(* CODESYS project e!C_Integration_Test_2.ECP

Project tree, tasks and I/O mapping:
  PFC_8206_PRO : 750-8206 PFC200 2ETH RS CAN DPS, WAGO, order no. 0750-8206, version 5.11.1.16
    application Application
      libraries: Util, * (System)
      task PLC_Task (cyclic, interval t#10ms, priority 14) calls PLC_PRG
      task VISU_TASK (cyclic, interval 100 ms, priority 15) calls VisuElems.Visu_Prg
      program PLC_PRG [ST]: Test2
      global variables NVL1_From8206
      declarations NVL1_From8203
      MODBUS/
        data type typFC_352_tcp
      global variables MODBUS
      visualisation Visu1
      image pool ImagePool8206
      global variables GNVL_RW_1
    DeviceAdapter
    Kbus : Kbus, WAGO, version 1.4.0.2
        unmapped channels: K-BUS diagnostics
      _8DI_8DO_24V_DC_0_5A : 0750-1506, WAGO, order no. 0750-1506, version 0.0.0.11
          settings: K-BUS Module slot index = 1
          input  LocalIn_Byte_1 AT %IB0 : BYTE  // _IN
          output LocalOut_Byte_1 AT %QB0 : BYTE  // _OUT
        DeviceAdapter
    MODBUS
      MODBUS : MODBUS, WAGO, order no. n/a, version 1.1.1.15
        _internal_1006_0001_Master : MODBUS Master, WAGO, order no. n/a, version 1.1.1.15
          _internal_1006_0001_IP : MODBUS IP Interface, WAGO, order no. n/a, version 1.1.1.15
              settings: IP settings.Address = '192.168.1.8'; Minimum Request Interval = 0 ms
            _internal_1006_0001_Remote_Slave : MODBUS Remote Slave, WAGO, order no. n/a, version 1.1.1.15
                settings: GeneratedChannel 100005.Cycle Time = 200 ms; GeneratedChannel 100005.Write Address = 512 Registers or Coils; GeneratedChannel 100005.Write Length = 1 Registers or Coils; Offset 100010 = 0; Slave address / Unit identifier = 1
                output Application.MODBUS.FC_352_tcp.dOut_1 : BOOL  // Mapping100020
    PROFIBUS
      PROFIBUS : PROFIBUS, WAGO, version 1.0.0.0
          settings: DT_Slot1_std:ARRAY[0..9] OF BYTE = 40; CT_Slot1_std:ARRAY[0..9] OF BYTE = 2; DT_Slot2_std:ARRAY[0..9] OF BYTE = 40; CT_Slot2_std:ARRAY[0..9] OF BYTE = 1
          input  To8206_ByteArray_1 : ARRAY[0..9] OF BYTE  // Slot1
          output From8206_ByteArray_1 : ARRAY[0..9] OF BYTE  // Slot2
    CANbus
      WAGO_CANopen_Manager : WAGO CANopen Manager, WAGO, version 3.5.4.10
          settings: ConfigVersion = 50659584
        _750_347m_V14 : 750-347m_V14, WAGO, order no. 750-347, version Revision=16#00000001, FileVersion=1.14
            settings: General Options.Reset Node = false; NODEIDSAVED = 4; SDO Timeout = 1000000; SubIndex for reset node = 0; Emergency-General Parameters.Emergency COBID = 16#00000084; Settings.COBID = 16#00000204; Settings.Transmission Type = 16#FF; Settings.available PDO-Parameter.Inhibit Time available = FALSE; Settings.available PDO-Parameter.Event Timer available = FALSE; Settings.Inhibit Time = 0; Settings.Event Timer = 0; Generic COBID = '$NODEID+16#0200'; Process by CANopenManager = TRUE; Settings.COBID = 16#00000184; Settings.Transmission Type = 16#FF; Settings.available PDO-Parameter.Inhibit Time available = TRUE; Settings.available PDO-Parameter.Event Timer available = TRUE; Settings.Inhibit Time = 0; Settings.Event Timer = 0; Generic COBID = '$NODEID+16#0180'; Process by CANopenManager = TRUE; WriteOutput8Bit : _75x_504_1.Index = 16#6200; WriteOutput8Bit : _75x_504_1.Subindex = 16#01; WriteOutput8Bit : _75x_504_1.ObjectLength = 8; ReadAnalogueInput16Bit : _75x_455_1.Index = 16#6401; ReadAnalogueInput16Bit : _75x_455_1.Subindex = 16#01; ReadAnalogueInput16Bit : _75x_455_1.ObjectLength = 16; ReadAnalogueInput16Bit : _75x_455_1.Index = 16#6401; ReadAnalogueInput16Bit : _75x_455_1.Subindex = 16#02; ReadAnalogueInput16Bit : _75x_455_1.ObjectLength = 16; ReadAnalogueInput16Bit : _75x_455_1.Index = 16#6401; ReadAnalogueInput16Bit : _75x_455_1.Subindex = 16#03; ReadAnalogueInput16Bit : _75x_455_1.ObjectLength = 16; ReadAnalogueInput16Bit : _75x_455_1.Index = 16#6401; ReadAnalogueInput16Bit : _75x_455_1.Subindex = 16#04; ReadAnalogueInput16Bit : _75x_455_1.ObjectLength = 16; SDO List.Set Guardtime.Index = 16#100C; SDO List.Set Guardtime.Subindex = 16#00; SDO List.Set Guardtime.Value = 16#00000000; SDO List.Set Guardtime.Size = 16;
              SDO List.Set Guardtime.AbortIfError = FALSE; SDO List.Set Guardtime.JumpToLine = FALSE; SDO List.Set Guardtime.Line = 0; SDO List.Set Lifetime.Index = 16#100D; SDO List.Set Lifetime.Subindex = 16#00; SDO List.Set Lifetime.Value = 16#00000000; SDO List.Set Lifetime.Size = 8; SDO List.Set Lifetime.AbortIfError = FALSE; SDO List.Set Lifetime.JumpToLine = FALSE; SDO List.Set Lifetime.Line = 0; SDO List.Disable Emcy CobID.Index = 16#1014; SDO List.Disable Emcy CobID.Subindex = 16#00; SDO List.Disable Emcy CobID.Value = 16#80000084; SDO List.Disable Emcy CobID.Size = 32; SDO List.Disable Emcy CobID.AbortIfError = FALSE; SDO List.Disable Emcy CobID.JumpToLine = FALSE; SDO List.Disable Emcy CobID.Line = 0; SDO List.Set Emcy CobID.Index = 16#1014; SDO List.Set Emcy CobID.Subindex = 16#00; SDO List.Set Emcy CobID.Value = 16#00000084; SDO List.Set Emcy CobID.Size = 32; SDO List.Set Emcy CobID.AbortIfError = FALSE; SDO List.Set Emcy CobID.JumpToLine = FALSE; SDO List.Set Emcy CobID.Line = 0; SDO List.Set Heartbeat Consumer.Index = 16#1016; SDO List.Set Heartbeat Consumer.Subindex = 16#01; SDO List.Set Heartbeat Consumer.Value = 0; SDO List.Set Heartbeat Consumer.Size = 32; SDO List.Set Heartbeat Consumer.AbortIfError = FALSE; SDO List.Set Heartbeat Consumer.JumpToLine = FALSE; SDO List.Set Heartbeat Consumer.Line = 0; SDO List.Set Heartbeat Consumer.Index = 16#1016; SDO List.Set Heartbeat Consumer.Subindex = 16#02; SDO List.Set Heartbeat Consumer.Value = 0; SDO List.Set Heartbeat Consumer.Size = 32; SDO List.Set Heartbeat Consumer.AbortIfError = FALSE; SDO List.Set Heartbeat Consumer.JumpToLine = FALSE; SDO List.Set Heartbeat Consumer.Line = 0; SDO List.Set Heartbeat Consumer.Index = 16#1016; SDO List.Set Heartbeat Consumer.Subindex = 16#03;
              SDO List.Set Heartbeat Consumer.Value = 0; SDO List.Set Heartbeat Consumer.Size = 32; SDO List.Set Heartbeat Consumer.AbortIfError = FALSE; SDO List.Set Heartbeat Consumer.JumpToLine = FALSE; SDO List.Set Heartbeat Consumer.Line = 0; SDO List.Set Heartbeat Consumer.Index = 16#1016; SDO List.Set Heartbeat Consumer.Subindex = 16#04; SDO List.Set Heartbeat Consumer.Value = 0; SDO List.Set Heartbeat Consumer.Size = 32; SDO List.Set Heartbeat Consumer.AbortIfError = FALSE; SDO List.Set Heartbeat Consumer.JumpToLine = FALSE; SDO List.Set Heartbeat Consumer.Line = 0; SDO List.Set Heartbeat Consumer.Index = 16#1016; SDO List.Set Heartbeat Consumer.Subindex = 16#05; SDO List.Set Heartbeat Consumer.Value = 0; SDO List.Set Heartbeat Consumer.Size = 32; SDO List.Set Heartbeat Consumer.AbortIfError = FALSE; SDO List.Set Heartbeat Consumer.JumpToLine = FALSE; SDO List.Set Heartbeat Consumer.Line = 0; SDO List.Set Heartbeat Producer.Index = 16#1017; SDO List.Set Heartbeat Producer.Subindex = 16#00; SDO List.Set Heartbeat Producer.Value = 16#00000000; SDO List.Set Heartbeat Producer.Size = 16; SDO List.Set Heartbeat Producer.AbortIfError = FALSE; SDO List.Set Heartbeat Producer.JumpToLine = FALSE; SDO List.Set Heartbeat Producer.Line = 0; SDO List.Disable PDO.Index = 16#1400; SDO List.Disable PDO.Subindex = 16#01; SDO List.Disable PDO.Value = 16#80000204; SDO List.Disable PDO.Size = 32; SDO List.Disable PDO.AbortIfError = FALSE; SDO List.Disable PDO.JumpToLine = FALSE; SDO List.Disable PDO.Line = 0; SDO List.Set transmission type.Index = 16#1400; SDO List.Set transmission type.Subindex = 16#02; SDO List.Set transmission type.Value = 16#FF; SDO List.Set transmission type.Size = 8; SDO List.Set transmission type.AbortIfError = FALSE; SDO List.Set transmission type.JumpToLine = FALSE; SDO List.Set transmission type.Line = 0;
              SDO List.Clear pdo mapping.Index = 16#1600; SDO List.Clear pdo mapping.Subindex = 16#00; SDO List.Clear pdo mapping.Value = 16#0; SDO List.Clear pdo mapping.Size = 8; SDO List.Clear pdo mapping.AbortIfError = FALSE; SDO List.Clear pdo mapping.JumpToLine = FALSE; SDO List.Clear pdo mapping.Line = 0; SDO List.Set Mapping.Index = 16#1600; SDO List.Set Mapping.Subindex = 16#01; SDO List.Set Mapping.Value = 16#62000108; SDO List.Set Mapping.Size = 32; SDO List.Set Mapping.AbortIfError = FALSE; SDO List.Set Mapping.JumpToLine = FALSE; SDO List.Set Mapping.Line = 0; SDO List.Set number of mappings.Index = 16#1600; SDO List.Set number of mappings.Subindex = 16#00; SDO List.Set number of mappings.Value = 16#01; SDO List.Set number of mappings.Size = 8; SDO List.Set number of mappings.AbortIfError = FALSE; SDO List.Set number of mappings.JumpToLine = FALSE; SDO List.Set number of mappings.Line = 0; SDO List.Set and enable COB-ID.Index = 16#1400; SDO List.Set and enable COB-ID.Subindex = 16#01; SDO List.Set and enable COB-ID.Value = 16#00000204; SDO List.Set and enable COB-ID.Size = 32; SDO List.Set and enable COB-ID.AbortIfError = FALSE; SDO List.Set and enable COB-ID.JumpToLine = FALSE; SDO List.Set and enable COB-ID.Line = 0; SDO List.Disable PDO.Index = 16#1800; SDO List.Disable PDO.Subindex = 16#01; SDO List.Disable PDO.Value = 16#80000184; SDO List.Disable PDO.Size = 32; SDO List.Disable PDO.AbortIfError = FALSE; SDO List.Disable PDO.JumpToLine = FALSE; SDO List.Disable PDO.Line = 0; SDO List.Set transmission type.Index = 16#1800; SDO List.Set transmission type.Subindex = 16#02; SDO List.Set transmission type.Value = 16#FF; SDO List.Set transmission type.Size = 8; SDO List.Set transmission type.AbortIfError = FALSE;
              SDO List.Set transmission type.JumpToLine = FALSE; SDO List.Set transmission type.Line = 0; SDO List.Set inhibit time.Index = 16#1800; SDO List.Set inhibit time.Subindex = 16#03; SDO List.Set inhibit time.Value = 16#0000; SDO List.Set inhibit time.Size = 16; SDO List.Set inhibit time.AbortIfError = FALSE; SDO List.Set inhibit time.JumpToLine = FALSE; SDO List.Set inhibit time.Line = 0; SDO List.Set event time.Index = 16#1800; SDO List.Set event time.Subindex = 16#05; SDO List.Set event time.Value = 16#0000; SDO List.Set event time.Size = 16; SDO List.Set event time.AbortIfError = FALSE; SDO List.Set event time.JumpToLine = FALSE; SDO List.Set event time.Line = 0; SDO List.Clear pdo mapping.Index = 16#1A00; SDO List.Clear pdo mapping.Subindex = 16#00; SDO List.Clear pdo mapping.Value = 16#0; SDO List.Clear pdo mapping.Size = 8; SDO List.Clear pdo mapping.AbortIfError = FALSE; SDO List.Clear pdo mapping.JumpToLine = FALSE; SDO List.Clear pdo mapping.Line = 0; SDO List.Set Mapping.Index = 16#1A00; SDO List.Set Mapping.Subindex = 16#01; SDO List.Set Mapping.Value = 16#64010110; SDO List.Set Mapping.Size = 32; SDO List.Set Mapping.AbortIfError = FALSE; SDO List.Set Mapping.JumpToLine = FALSE; SDO List.Set Mapping.Line = 0; SDO List.Set Mapping.Index = 16#1A00; SDO List.Set Mapping.Subindex = 16#02; SDO List.Set Mapping.Value = 16#64010210; SDO List.Set Mapping.Size = 32; SDO List.Set Mapping.AbortIfError = FALSE; SDO List.Set Mapping.JumpToLine = FALSE; SDO List.Set Mapping.Line = 0; SDO List.Set Mapping.Index = 16#1A00; SDO List.Set Mapping.Subindex = 16#03; SDO List.Set Mapping.Value = 16#64010310;
              SDO List.Set Mapping.Size = 32; SDO List.Set Mapping.AbortIfError = FALSE; SDO List.Set Mapping.JumpToLine = FALSE; SDO List.Set Mapping.Line = 0; SDO List.Set Mapping.Index = 16#1A00; SDO List.Set Mapping.Subindex = 16#04; SDO List.Set Mapping.Value = 16#64010410; SDO List.Set Mapping.Size = 32; SDO List.Set Mapping.AbortIfError = FALSE; SDO List.Set Mapping.JumpToLine = FALSE; SDO List.Set Mapping.Line = 0; SDO List.Set number of mappings.Index = 16#1A00; SDO List.Set number of mappings.Subindex = 16#00; SDO List.Set number of mappings.Value = 16#04; SDO List.Set number of mappings.Size = 8; SDO List.Set number of mappings.AbortIfError = FALSE; SDO List.Set number of mappings.JumpToLine = FALSE; SDO List.Set number of mappings.Line = 0; SDO List.Set and enable COB-ID.Index = 16#1800; SDO List.Set and enable COB-ID.Subindex = 16#01; SDO List.Set and enable COB-ID.Value = 16#00000184; SDO List.Set and enable COB-ID.Size = 32; SDO List.Set and enable COB-ID.AbortIfError = FALSE; SDO List.Set and enable COB-ID.JumpToLine = FALSE; SDO List.Set and enable COB-ID.Line = 0; ConfigVersion = 50659584
          DeviceAdapter
          _75x_504_1 : 75x-504, WAGO, order no. 75x-504, version Revision=16#00000001, FileVersion=1.14
              settings: Number of Params = 1; WriteOutput8Bit : _75x_504_1.Index = 16#6200; WriteOutput8Bit : _75x_504_1.Subindex = 16#01; WriteOutput8Bit : _75x_504_1.Startbit = 0; WriteOutput8Bit : _75x_504_1.Endbit = 3
              output Application.PLC_PRG.CANopen_To347_DO_1 : BOOL  // WriteOutput8Bit : _75x_504_1.Bit0
              unmapped channels: WriteOutput8Bit : _75x_504_1
          _75x_455_1 : 75x-455, WAGO, order no. 75x-455, version Revision=16#00000001, FileVersion=1.14
              settings: Number of Params = 4; ReadAnalogueInput16Bit : _75x_455_1.Index = 16#6401; ReadAnalogueInput16Bit : _75x_455_1.Subindex = 16#01; ReadAnalogueInput16Bit : _75x_455_1.Startbit = 0; ReadAnalogueInput16Bit : _75x_455_1.Endbit = 15; ReadAnalogueInput16Bit : _75x_455_1.Index = 16#6401; ReadAnalogueInput16Bit : _75x_455_1.Subindex = 16#02; ReadAnalogueInput16Bit : _75x_455_1.Startbit = 0; ReadAnalogueInput16Bit : _75x_455_1.Endbit = 15; ReadAnalogueInput16Bit : _75x_455_1.Index = 16#6401; ReadAnalogueInput16Bit : _75x_455_1.Subindex = 16#03; ReadAnalogueInput16Bit : _75x_455_1.Startbit = 0; ReadAnalogueInput16Bit : _75x_455_1.Endbit = 15; ReadAnalogueInput16Bit : _75x_455_1.Index = 16#6401; ReadAnalogueInput16Bit : _75x_455_1.Subindex = 16#04; ReadAnalogueInput16Bit : _75x_455_1.Startbit = 0; ReadAnalogueInput16Bit : _75x_455_1.Endbit = 15
              input  Application.PLC_PRG.CANopen_From347_AI_1 : WORD  // ReadAnalogueInput16Bit : _75x_455_1
              unmapped channels: ReadAnalogueInput16Bit : _75x_455_1, ReadAnalogueInput16Bit : _75x_455_1, ReadAnalogueInput16Bit : _75x_455_1
    Serial
      COM1 : COM1, WAGO, version 0.0.0.19
  PFC_8203_CAN : 750-8203 PFC200 2ETH CAN, WAGO, order no. 0750-8203, version 5.11.1.16
    application Application
      task PLC_Task (cyclic, interval t#10ms, priority 14) calls PLC_PRG
      program PLC_PRG [ST]: Test2
      declarations NVL1_From8206
      global variables NVL1_From8203
      global variables GNVL_RW_1
    DeviceAdapter
    Kbus : Kbus, WAGO, version 1.4.0.2
        unmapped channels: K-BUS diagnostics
      _8_DO_24_V_DC_0_5A : 0750-0530, WAGO, order no. 0750-0530, version 0.0.0.15
          settings: K-BUS Module slot index = 2
          unmapped channels: _OUT
        DeviceAdapter
      _8_DI_24_V_DC_3_0ms : 0750-0430, WAGO, order no. 0750-0430, version 0.0.0.14
          settings: K-BUS Module slot index = 1
          unmapped channels: _IN
        DeviceAdapter
    MODBUS
      MODBUS : MODBUS, WAGO, order no. n/a, version 1.1.1.15
    CANbus
  FC_352 : 750-352, WAGO, order no. 0750-0352, version 0.0.0.9
    DeviceAdapter
    Kbus : Kbus, WAGO, version 0.0.0.101
        unmapped channels: K-BUS diagnostics
      _4_DO_Generic : 075x-4DO, WAGO, order no. 075x-4DO, version 0.0.0.13
          settings: K-BUS Module slot index = 1
          unmapped channels: _OUT
        DeviceAdapter
  Generic_PROFIBUS_Master : ThirdParty Profibus Master, WAGO, order no. GenericProfibusMaster, version 1.0.0.3
    DeviceAdapter
    Profibus
  libraries: WagoVisuIcons, 1.0.0.8 (WAGO)
  text list GlobalTextList
  5ce3da45-db07-42e7-a21c-a00fff4ed8f6|C:\MySD\Dropbox (Wago Norge)\Torgeir\Development\Customer_Projects\Eltorque\Eltorque_QT250.gif
*)

// PFC_8206_PRO/Application/MODBUS/typFC_352_tcp
TYPE typFC_352_tcp:
STRUCT
	dOut_1: BOOL;
END_STRUCT
END_TYPE

// PFC_8206_PRO/Application/NVL1_From8206
VAR_GLOBAL
	NV1_From8206_ByteArray : ARRAY[0..9] OF BYTE;
END_VAR

// PFC_8203_CAN/Application/NVL1_From8206
//This gobal variable list is received via the network.
//Sender: NVL1_From8206 [PFC_8206_PRO: PLC Logic: Application]
//Protocol: UDP

VAR_GLOBAL
	NV1_From8206_ByteArray : ARRAY[0..9] OF BYTE;
END_VAR

// PFC_8203_CAN/Application/NVL1_From8203
VAR_GLOBAL
	NV1_From8203_ByteArray : ARRAY[0..9] OF BYTE;
END_VAR

// PFC_8206_PRO/Application/NVL1_From8203
//This gobal variable list is received via the network.
//Sender: NVL1_From8203 [PFC_8203_CAN: PLC Logic: Application]
//Protocol: UDP

VAR_GLOBAL
	NV1_From8203_ByteArray : ARRAY[0..9] OF BYTE;
END_VAR

// PFC_8206_PRO/Application/MODBUS
VAR_GLOBAL
	FC_352_tcp: typFC_352_tcp;
END_VAR

// PFC_8206_PRO/Application/GNVL_RW_1
VAR_GLOBAL
	wFra8203_Test_1: WORD;
	wFra8206_Test_1: WORD;
END_VAR

// PFC_8203_CAN/Application/GNVL_RW_1
VAR_GLOBAL
	wFra8203_Test_1: WORD;
	wFra8206_Test_1: WORD;
END_VAR

// PFC_8206_PRO/Application/PLC_PRG
PROGRAM PLC_PRG
VAR
	CANopen_From347_AI_1: WORD;
	CANopen_To347_DO_1: BOOL;
	BLINK1: BLINK := (ENABLE := TRUE, TIMELOW := TIME#1s0ms, TIMEHIGH := TIME#1s0ms);
	Lampe1: BOOL;
	Knapp1: BOOL;
	VisuInput: INT;

	tidhoy: TIME := T#2s;
	tidlav: TIME := T#2s;
	BLINK2: BLINK;
	blink2ut: BOOL;

	GVNVL_1_trigger : BOOL;

END_VAR



BLINK1(ENABLE:= , TIMELOW:= , TIMEHIGH:= , OUT=> );


LocalOut_Byte_1 := To8206_ByteArray_1[0];
From8206_ByteArray_1[0] := LocalIn_Byte_1;
NV1_From8206_ByteArray := To8206_ByteArray_1;
NV1_From8203_ByteArray;


CANopen_From347_AI_1;
CANopen_To347_DO_1 := BLINK1.OUT;


FC_352_tcp.dOut_1 := BLINK1.OUT;

Lampe1 := Knapp1;

wFra8203_Test_1 := wFra8203_Test_1 + 1;
wFra8206_Test_1 := wFra8206_Test_1 + 1;
GVNVL_1_trigger := BLINK1.OUT;

Test2();

ACTION Test2:
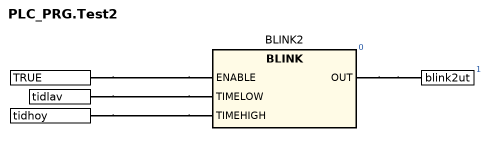
BLINK2(ENABLE := TRUE, TIMELOW := tidlav, TIMEHIGH := tidhoy); // BLINK
blink2ut := BLINK2.OUT;
END_ACTION

END_PROGRAM

// PFC_8203_CAN/Application/PLC_PRG
PROGRAM PLC_PRG
VAR
	GVNVL_1_trigger : BOOL;
	wFra8203_Test_1_tmp: WORD;
	wFra8206_Test_1_tmp: WORD;
END_VAR

NV1_From8203_ByteArray := NV1_From8206_ByteArray;

wFra8203_Test_1_tmp := wFra8203_Test_1;
wFra8206_Test_1_tmp := wFra8206_Test_1;
GVNVL_1_trigger;

Test2();

ACTION Test2:

END_ACTION

END_PROGRAM

// PFC_8206_PRO/Application/Visu1
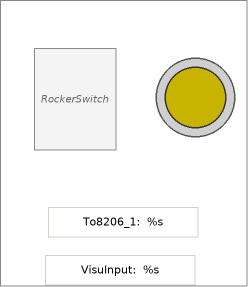
VISUALIZATION Visu1  // 248x287
    Lamp1 (145,51 101x93), variable: PLC_PRG.Lampe1, style: Lamp-Lamp1-Yellow
    RockerSwitch (34,48 82x102), variable: PLC_PRG.Knapp1, behaviour: TOGGLE, style: Switch-RockerSwitch-Gray
    Textfield (48,207 150x30), "To8206_1: %s", text variable: To8206_ByteArray_1[0]
    Textfield (45,255 150x30), "VisuInput: %s", text variable: PLC_PRG.VisuInput
        OnMouseDown: write the text variable via Edit
END_VISUALIZATION
